(* IEC 61131-3 sources: CodesysPractice/Lessons/Lesson1/st, 7 files *)

(* ---- DUT.st ---- *)
(* =====================================================================
   对象类型 : DUT            对象名 : DUT
   项目     : Lesson1
   角色     : 全工程唯一的自定义类型表，分两个层次：
              【领域类型】Axis（一根轴）、Cmd（一条命令）—— 业务的语言；
              【报文格式】AxisInfo（PLC 发给上位机的帧）—— 线上的字节合同。
              Cmd 同时就是上行帧（命令即报文）；AxisInfo 只是输出报文，
              不是与 Axis / Cmd 并列的领域概念。

   报文布局（pack_mode=1，双端 x86/x64 小端，内存拷贝即协议）:
      Cmd    30 字节 : bType(1) bSub(1) nLen(1) aParam[3]×AxisParam(27)
      AxisParam 9 字节 : bAxis(1) rPos(4) rVel(4)
      Axis   13 字节 : rActPos(4) rTargetPos(4) rVelocity(4) xMoving(1)
      AxisInfo 45 字节 : wResult(2) nAckSeq(4) aAxis[3]×Axis(39)

   创建方法 : Application 右键 -> 添加对象 -> DUT -> 名称 DUT
              -> 类型选"结构体"（多个结构体可放在同一个 DUT 对象里）。
   粘贴方法 : 本文件整段照粘（编辑器自带的外壳整段替换）。
   ===================================================================== *)

// ==================== 领域类型 ====================

// ---- 一根轴：设定 + 实际的全部家当 ----
{attribute 'pack_mode' := '1'}
TYPE Axis :
STRUCT
    rActPos    : REAL;   // 实际位置
    rTargetPos : REAL;   // 目标位置（最近一次 MoveTo 的设定）
    rVelocity  : REAL;   // 速度（最近一次 MoveTo 的设定）
    xMoving    : BOOL;   // TRUE=运动中，FALSE=Idle
END_STRUCT
END_TYPE

// ---- 一路轴参数（CMD_CONTENT 的元素）：轴号 + 位置 + 速度 ----
{attribute 'pack_mode' := '1'}
TYPE AxisParam :
STRUCT
    bAxis : BYTE;    // 轴号：1=X 2=Y 3=Z（即 GVL.aAxis 的下标）
    rPos  : REAL;    // MOVE 目标位置（STOP 时不用）
    rVel  : REAL;    // MOVE 速度，必须 > 0（STOP 时不用）
END_STRUCT
END_TYPE

// ---- 一条命令：上位机 -> PLC，同时就是上行帧，30 字节 ----
// 分层：命令头(bType) + 子命令(bSub) + 参数数组(aParam + 有效个数 nLen)。
// 一帧可携带多路轴参数，一次命令多根轴；每路自带轴号，顺序无关。
{attribute 'pack_mode' := '1'}
TYPE Cmd :
STRUCT
    bType  : BYTE;                      // 命令头：取值见 GVL 常量 CMD_MOVE / CMD_STOP
    bSub   : BYTE;                      // 子命令：预留，现填 0（将来如 MOVE 的绝对/相对）
    nLen   : BYTE;                      // aParam 里的有效路数：1..3
    aParam : ARRAY[1..3] OF AxisParam;  // 参数数组，只有前 nLen 路有效
END_STRUCT
END_TYPE

// ==================== 报文格式 ====================

// ---- 汇报帧：PLC -> 上位机，45 字节 ----
// 只是"PLC 发出的电报"：最近一条命令的结果 + 三轴现状。
// 回执序号变化立即发一帧，否则每 200ms 发一帧 —— 两种场合发同一个结构。
{attribute 'pack_mode' := '1'}
TYPE AxisInfo :
STRUCT
    wResult : WORD;                  // 最近一条命令的结果码（0=OK，其余见 GVL 结果码）
    nAckSeq : UDINT;                 // 回执序号：上位机靠它的变化识别"新回执"
    aAxis   : ARRAY[1..3] OF Axis;   // 三轴现状
END_STRUCT
END_TYPE

(* ---- GVL.st ---- *)
(* =====================================================================
   对象类型 : GVL            对象名 : GVL
   项目     : Lesson1
   角色     : 全工程唯一的全局变量表，分两层：
              【领域数据】三根轴、当前命令 —— 业务的语言；
              【配套机制】命令的处理结果、跨任务序号握手 —— 实现细节。
              纪律：一个变量只有一个写者。
   创建方法 : Application 右键 -> 添加对象 -> 全局变量列表（GVL）-> 名称 GVL。
   粘贴方法 : 本文件整段照粘（编辑器自带的 VAR_GLOBAL...END_VAR 外壳整段替换，
              注意本文件有两个 VAR_GLOBAL 块，都要粘进去）。
   ===================================================================== *)
{attribute 'qualified_only'}
VAR_GLOBAL CONSTANT
    // ==== 命令字：Cmd.bType 的合法取值 ====
    CMD_MOVE    : BYTE := 1;
    CMD_STOP    : BYTE := 2;

    // ==== 结果码：全工程唯一出处。AxisInfo.wResult 就是这里的值，
    //      上位机按码判错 ====
    OK          : WORD := 0;      // 成功
    UNKNOWN_CMD : WORD := 1001;   // 命令字不认识（只认 CMD_MOVE / CMD_STOP）
    BAD_AXIS    : WORD := 1002;   // 轴号不是 1..3
    BAD_PARAM   : WORD := 1003;   // 参数非法（如速度 <= 0）
    SOCK_CREATE : WORD := 9001;   // 监听套接字创建失败
    SOCK_BIND   : WORD := 9002;   // 端口绑定失败（最常见：端口被占用）
    SOCK_LISTEN : WORD := 9003;   // listen 失败
END_VAR

VAR_GLOBAL
    // ==== 领域数据 ====
    aAxis   : ARRAY[1..3] OF Axis;  // 三根轴：下标即轴号 1=X / 2=Y / 3=Z
                                    // （MainTask 写，CommTask 读去组 AxisInfo）
    stCmd   : Cmd;                  // 当前命令（CommTask 收帧写入，MainTask 处理）

    // ==== stCmd 的配套机制（跨任务握手，实现细节，不是领域概念）====
    // 规则：CommTask 凑满一帧 -> stCmd 已被 FB_TcpServer 写好 -> nCmdSeq +1；
    //      MainTask 看到 nCmdSeq <> nAckSeq 就处理，处理完写 wResult、
    //      把 nAckSeq 对齐 nCmdSeq。
    // 单命令槽：上一帧没被取走时会被新帧覆盖。命令是人手速发的，骨架阶段够用；
    //          将来接自动上位机时换命令队列。
    wResult : WORD;             // stCmd 的处理结果（MainTask 写）
    nCmdSeq : UDINT := 0;       // 命令序号，CommTask 每收满一帧 +1；回绕到 0 也安全
    nAckSeq : UDINT := 0;       // 回执序号，MainTask 处理完对齐 nCmdSeq
END_VAR

(* ---- FB_CmdHandler.st ---- *)
(* =====================================================================
   对象类型 : POU（FB，语言 ST）   对象名 : FB_CmdHandler
   项目     : Lesson1
   角色     : 命令处理：解析当前命令（GVL.stCmd），分发到具体的处理者。
              它只懂协议 —— 命令字合法吗、路数合法吗、轴号合法吗；不懂业务。
              MOVE / STOP 是轴命令，业务在轴的方法（MoveTo / Stop）里；
              将来命令集合扩张（新 bType、bSub 取值、非轴命令）时，
              新增对应的处理类、加分支即可，本类结构不变。
              多路命令采用两遍法：先整体校验，再逐路执行 ——
              要么全执行，要么全不执行，不存在"动了一半"。
   协议     : bType = GVL.CMD_MOVE / GVL.CMD_STOP；bSub 预留填 0
              nLen  = 1..3（aParam 的有效路数）
              每路：bAxis = 1..3；MOVE 要求 rVel > 0（轴自己也会再判一道）
   创建方法 : Application 右键 -> 添加对象 -> POU -> 名称 FB_CmdHandler
              -> 类型选"功能块"（Function Block）-> 实现语言选 ST。
   粘贴方法 : 跳过下面第一行对象头（FUNCTION_BLOCK xxx），声明区（各 VAR 块）
              粘到编辑器上半部，"实现区"分隔线以下的内容粘到下半部。
   ===================================================================== *)
FUNCTION_BLOCK FB_CmdHandler
VAR_INPUT
    stCmd   : Cmd;                          // 待处理的当前命令
END_VAR
VAR_IN_OUT
    aAxis   : ARRAY[1..3] OF FB_SimAxis;    // 分发目标：命令最终作用在轴上
END_VAR
VAR_OUTPUT
    wResult : WORD;                         // 处理结果码：GVL.OK 或结果码
END_VAR
VAR
    i       : INT;
    nAx     : INT;
END_VAR
(* ---------------- 实现区（以下粘到 POU 编辑器下半部） ---------------- *)
// 默认成功，走到哪步出错在哪步盖结果码
wResult := GVL.OK;

// --- 命令字（协议级校验）---
IF (stCmd.bType <> GVL.CMD_MOVE) AND (stCmd.bType <> GVL.CMD_STOP) THEN
    wResult := GVL.UNKNOWN_CMD;
    RETURN;
END_IF

// --- 有效路数 ---
IF (stCmd.nLen < 1) OR (stCmd.nLen > 3) THEN
    wResult := GVL.BAD_PARAM;
    RETURN;
END_IF

// --- 第一遍：整体校验全部路数（轴号；MOVE 还要速度 > 0）---
// 任何一路非法 -> 整体拒绝，一路都不执行
FOR i := 1 TO TO_INT(stCmd.nLen) DO
    IF (stCmd.aParam[i].bAxis < 1) OR (stCmd.aParam[i].bAxis > 3) THEN
        wResult := GVL.BAD_AXIS;
        RETURN;
    END_IF
    IF (stCmd.bType = GVL.CMD_MOVE) AND (stCmd.aParam[i].rVel <= 0) THEN
        wResult := GVL.BAD_PARAM;
        RETURN;
    END_IF
END_FOR

// --- 第二遍：逐路分发执行（校验已过，此处必成功）---
FOR i := 1 TO TO_INT(stCmd.nLen) DO
    nAx := TO_INT(stCmd.aParam[i].bAxis);
    CASE stCmd.bType OF
        GVL.CMD_MOVE:
            wResult := aAxis[nAx].MoveTo(stCmd.aParam[i].rPos,
                                         stCmd.aParam[i].rVel);
        GVL.CMD_STOP:
            aAxis[nAx].Stop();
    END_CASE
END_FOR

(* ---- FB_SimAxis.st ---- *)
(* =====================================================================
   对象类型 : POU（FB，语言 ST，带 2 个方法）   对象名 : FB_SimAxis
   项目     : Lesson1
   角色     : 仿真轴：恒速点位 + 立即停止。轴是对象：
              行为是方法（MoveTo / Stop），本体每周期只做积分更新。
              参数合法性（速度 > 0）由轴自己判 —— 那是轴的业务，
              不是协议的事。换真轴时方法内部改调 MC_MoveAbsolute /
              MC_Stop，调用侧零改动。
   为什么自写而不上 SoftMotion：架子阶段要的是"一定跑得起来"。虚拟轴也要
              装 SoftMotion、配三组轴对象，把通信架子的首跑拖进运动控制
              的泥潭；接口设计好，后面换芯不动架。
   创建方法 : Application 右键 -> 添加对象 -> POU -> 名称 FB_SimAxis
              -> 类型选"功能块"（Function Block）-> 实现语言选 ST。
              然后右键 FB_SimAxis -> 添加对象 -> 方法（Method）：
              名 MoveTo、返回类型 WORD、语言 ST；名 Stop、无返回类型、语言 ST。
   粘贴方法 : FB 本体：跳过第一行对象头，VAR 块粘到上半部，"本体实现区"
              分隔线以下粘到下半部。★ 两个 METHOD 分隔线以下的内容
              **不要粘进 FB**（FB 里出现 METHOD 关键字会报"未预期的语句"）——
              方法是挂在 FB 下的独立子对象，逐节粘进对应的方法编辑器：
              跳过该节的 METHOD 对象头（IDE 按创建对话框自动生成），
              VAR 块粘上半部，实现粘下半部。
   ===================================================================== *)
FUNCTION_BLOCK FB_SimAxis
VAR_INPUT
    rCycleTime : REAL := 0.01;   // 调用任务的周期（秒），由调用方按任务配置填
END_VAR
VAR_OUTPUT
    rActPos    : REAL;           // 实际位置
    rTargetPos : REAL;           // 目标位置（最近一次 MoveTo 的设定）
    rVelocity  : REAL;           // 速度（最近一次 MoveTo 的设定）
    xMoving    : BOOL;           // TRUE=运动中
END_VAR
VAR
    rDir  : REAL := 1.0;         // 运动方向（+1/-1），MoveTo 时设定
    rStep : REAL;                // 本周期的步进量
END_VAR
(* ---------------- 本体实现区（粘到 FB 编辑器下半部） ---------------- *)
// 本体每周期只做一件事：恒速积分，到点钳位（防过冲）
IF xMoving THEN
    rStep := rVelocity * rCycleTime * rDir;
    IF ((rDir > 0) AND ((rActPos + rStep) >= rTargetPos)) OR
       ((rDir < 0) AND ((rActPos + rStep) <= rTargetPos)) THEN
        rActPos := rTargetPos;
        xMoving := FALSE;                        // 到位
    ELSE
        rActPos := rActPos + rStep;
    END_IF
END_IF

(* ============ METHOD MoveTo（独立子对象，不要粘进 FB 本体！） ============ *)
METHOD MoveTo : WORD
VAR_INPUT
    rPos : REAL;   // 目标位置
    rVel : REAL;   // 速度，必须 > 0
END_VAR
(* ---- MoveTo 实现 ---- *)
// 返回值是 GVL 结果码；运动中再来 = 改目标
MoveTo := GVL.OK;
IF rVel <= 0 THEN
    MoveTo := GVL.BAD_PARAM;
    RETURN;
END_IF
rTargetPos := rPos;
rVelocity  := rVel;
IF rTargetPos = rActPos THEN
    xMoving := FALSE;                            // 已经在点上
ELSE
    xMoving := TRUE;
    IF rTargetPos > rActPos THEN
        rDir := 1.0;
    ELSE
        rDir := -1.0;
    END_IF
END_IF

(* ============ METHOD Stop（独立子对象，不要粘进 FB 本体！） ============ *)
METHOD Stop
(* ---- Stop 实现 ---- *)
// 立即停止
xMoving := FALSE;

(* ---- FB_TcpServer.st ---- *)
(* =====================================================================
   对象类型 : POU（FB，语言 ST）   对象名 : FB_TcpServer
   项目     : Lesson1
   运行目标 : CODESYS Control Win V3 x64（64 位！）
   角色     : TCP 服务器封装（SysSocket 库）：监听 -> 接单客户端 ->
              收字节凑成定长帧 / 把一帧发出去。协议内容它一概不懂，
              只认识帧长度 —— 这就是"协议层"和"通道层"的分界。
   纪律     : 全部 socket 调用都是非阻塞的（FIONBIO），
              绝不许把 CommTask 卡死在对端的沉默上。
   注意     : 定长帧没有同步头 —— 对端发来的字节数一旦错位就会永久错位。
              骨架双方都是自己人（配套上位机），不处理；接陌生对端时
              要加帧头 + 长度 + CRC（已记入项目 README 的扩展点）。

   —— 为什么用 SysSocket 而不是 SysSockets23 ——
   旧的 SysSockets23（3.5.13.0）是 32 位专用库，在 x64 设备上编译直接报
   C0338（该库不支持 64 位应用程序）。现役的 **SysSocket**（3.5.19.0）
   是 32/64 位通用版，本文件按它的实际签名编写。

   创建方法 : Application 右键 -> 添加对象 -> POU -> 名称 FB_TcpServer
              -> 类型选"功能块"（Function Block）-> 实现语言选 ST。
   库       : Library Manager -> Add Library -> 搜 syssocket -> 选 **SysSocket**
              （3.5.19.0）。★ 不要选 SysSocket23（32 位专用），
              也不要选 SysSocket2（另一套已废弃的 2.x 接口）。
              加好后把旧的 SysSockets23 从 Library Manager 里删掉。
   粘贴方法 : 跳过下面第一行对象头（FUNCTION_BLOCK xxx），声明区（各 VAR 块）
              粘到编辑器上半部，"实现区"分隔线以下的内容粘到下半部。
   ===================================================================== *)
FUNCTION_BLOCK FB_TcpServer
VAR_INPUT
    xEnable : BOOL := TRUE;      // FALSE 时关闭连接与监听，回到空闲
    nPort   : UINT := 12000;
    pRxBuf  : POINTER TO BYTE;   // 收帧目标：凑满 nRxSize 字节 = 一帧
    nRxSize : UINT;              // 收帧长度（调用方传 SIZEOF(命令结构体)）
    pTxBuf  : POINTER TO BYTE;   // 待发的一帧
    nTxSize : UINT;              // 发帧长度
    xSend   : BOOL;              // 上升沿把 pTxBuf 指向的 nTxSize 字节发出去
END_VAR
VAR_OUTPUT
    xClientConnected : BOOL;
    xFrameReady : BOOL;          // 本周期凑满一帧（pRxBuf 内容已更新），保持一个周期
    bError      : BOOL;          // 保持型：建监听失败才置位，码见 GVL.SOCK_*
    nErrorID    : WORD;
END_VAR
VAR
    eState     : INT := 0;       // 0=空闲 / 1=监听中 / 2=已连接；不出本 FB，故不建枚举
    hListen    : RTS_IEC_HANDLE := RTS_INVALID_HANDLE;
    hClient    : RTS_IEC_HANDLE := RTS_INVALID_HANDLE;
    hNew       : RTS_IEC_HANDLE;
    sockAddr    : SOCKADDRESS;   // 本机监听地址
    sockAddrCli : SOCKADDRESS;   // accept 回写的客户端地址（内容不用，签名要指针）
    diAddrLen   : DINT;          // sockAddrCli 的长度（accept 的入/出参）
    resOp      : RTS_IEC_RESULT; // create / bind / listen / accept 的返回码
    resRecv    : RTS_IEC_RESULT; // recv 的返回码：区分"对端关闭"与"暂无数据"
    resSend    : RTS_IEC_RESULT;
    diNonBlock : DINT := 1;      // FIONBIO 参数：1 = 非阻塞
    diReuse    : DINT := 1;      // SO_REUSEADDR 参数：1 = 允许地址复用
    diRet      : __XINT;         // recv 返回值。__XINT = 平台相关整型（x64 下 64 位），
                                 // 必须用 __XINT 接，用 DINT 接在 x64 上报类型错
    diSent     : __XINT;         // send 返回值：<=0 视为发送失败（对端已死）
    diRxCnt    : INT;            // 本帧已收字节数（兼作写入偏移；指针运算用 INT 最稳）
    xBufSize   : __XINT;         // recv / send 的缓冲长度入参：类型必须和形参一致（__XINT），
                                 // 先把长度算进这个变量，实参里就不做类型转换
    xSendPrev  : BOOL;
END_VAR
VAR CONSTANT
    // SysSocket 函数的成功返回码 = 0。
    // 不直接写库常量 ERR_OK：它由库的依赖链带出，库版本一变就可能"没有定义标识符"。
    // 用本地常量最稳，语义一样。
    SOCK_OK : RTS_IEC_RESULT := 0;
    // x64 下 SysSocket 出错时返回的非法句柄是 16#FFFFFFFFFFFFFFFF
    // （Windows 的 INVALID_SOCKET），与 RTS_INVALID_HANDLE
    // （16#00000000FFFFFFFF）不相等！create / accept 拿到返回值后先归一成
    // RTS_INVALID_HANDLE，否则空 accept 会被当成接到了客户端
    // （假连接死循环：发送失败 -> 回监听 -> 又假 accept，真客户端进不来）。
    HANDLE_INVALID : RTS_IEC_HANDLE := 16#FFFFFFFFFFFFFFFF;
END_VAR
(* ---------------- 实现区（以下粘到 POU 编辑器下半部） ---------------- *)
xFrameReady := FALSE;

// --- 使能撤掉：关干净回空闲 ---
IF NOT xEnable THEN
    IF (hClient <> RTS_INVALID_HANDLE) AND (hClient <> 0) THEN
        SysSockClose(hClient);
        hClient := RTS_INVALID_HANDLE;
    END_IF
    IF (hListen <> RTS_INVALID_HANDLE) AND (hListen <> 0) THEN
        SysSockClose(hListen);
        hListen := RTS_INVALID_HANDLE;
    END_IF
    eState := 0;
    xClientConnected := FALSE;
    diRxCnt := 0;
END_IF

CASE eState OF

    // ---------------------------------------------------------------
    0:  // 空闲：建立监听
        bError := FALSE;
        nErrorID := GVL.OK;
        IF xEnable THEN
            // SysSockCreate(iAddressFamily : INT, diType : DINT, diProtocol : DINT,
            //               pResult : POINTER TO RTS_IEC_RESULT) : RTS_IEC_HANDLE
            hListen := SysSockCreate(SOCKET_AF_INET, SOCKET_STREAM, SOCKET_IPPROTO_TCP,
                                     ADR(resOp));
            IF hListen = HANDLE_INVALID THEN
                hListen := RTS_INVALID_HANDLE;   // 归一非法句柄，见 HANDLE_INVALID 注释
            END_IF
            IF (hListen = RTS_INVALID_HANDLE) OR (hListen = 0) THEN
                bError := TRUE;
                nErrorID := GVL.SOCK_CREATE;
                hListen := RTS_INVALID_HANDLE;
            ELSE
                // 非阻塞：accept / recv 没有事件时立即返回，不卡任务
                // SysSockIoctl(hSocket, diCommand : DINT, pdiParameter : POINTER TO DINT)
                SysSockIoctl(hListen, SOCKET_FIONBIO, ADR(diNonBlock));
                // 允许地址复用：调试时反复"下载/运行"不会报端口被占用（9002）
                // SysSockSetOption(hSocket, diLevel : DINT, diOption : DINT,
                //                  pdiOptionValue : POINTER TO DINT, diOptionLen : DINT)
                SysSockSetOption(hListen, SOCKET_SOL, SOCKET_SO_REUSEADDR,
                                 ADR(diReuse), SIZEOF(diReuse));

                sockAddr.sin_family      := SOCKET_AF_INET;      // INT，直接赋值，不要 TO_INT
                // 端口必须转成网络字节序；显式 WORD 转型避免 UINT->WORD 的隐式转换告警
                sockAddr.sin_port        := SysSockHtons(TO_WORD(nPort));
                sockAddr.sin_addr.ulAddr := SOCKET_INADDR_ANY;   // 0.0.0.0，本机所有网卡都接

                // SysSockBind(hSocket, pSockAddr : POINTER TO SOCKADDRESS,
                //             diSockAddrSize : DINT) : RTS_IEC_RESULT
                IF SysSockBind(hListen, ADR(sockAddr), SIZEOF(sockAddr)) <> SOCK_OK THEN
                    bError := TRUE;
                    nErrorID := GVL.SOCK_BIND;
                // SysSockListen(hSocket, diMaxConnections : DINT) : RTS_IEC_RESULT
                ELSIF SysSockListen(hListen, 1) <> SOCK_OK THEN
                    bError := TRUE;
                    nErrorID := GVL.SOCK_LISTEN;
                ELSE
                    eState := 1;
                END_IF
                IF bError THEN
                    SysSockClose(hListen);
                    hListen := RTS_INVALID_HANDLE;
                END_IF
            END_IF
        END_IF

    // ---------------------------------------------------------------
    1:  // 监听中：非阻塞 accept，接到就进已连接
        // SysSockAccept(hSocket, pSockAddr : POINTER TO SOCKADDRESS,
        //               pdiSockAddrSize : POINTER TO DINT,
        //               pResult) : RTS_IEC_HANDLE
        // 注意：x64 版不接受空指针（0），必须传真实的地址变量和长度变量
        diAddrLen := SIZEOF(sockAddrCli);
        hNew := SysSockAccept(hListen, ADR(sockAddrCli), ADR(diAddrLen), ADR(resOp));
        IF hNew = HANDLE_INVALID THEN
            hNew := RTS_INVALID_HANDLE;          // 归一非法句柄，见 HANDLE_INVALID 注释
        END_IF
        IF (hNew <> RTS_INVALID_HANDLE) AND (hNew <> 0) THEN
            hClient := hNew;
            SysSockIoctl(hClient, SOCKET_FIONBIO, ADR(diNonBlock));
            diRxCnt := 0;
            xClientConnected := TRUE;
            eState := 2;
        END_IF

    // ---------------------------------------------------------------
    2:  // 已连接：收字节凑帧 / 发一帧
        // -- 收：往调用方的帧缓冲里续字节，凑满 nRxSize 即一帧 --
        IF (pRxBuf <> 0) AND (nRxSize > 0) THEN
            // SysSockRecv(hSocket, pbyBuffer : POINTER TO BYTE, diBufferSize : __XINT,
            //             diFlags : DINT, pResult) : __XINT
            // flags 传 NONE：非阻塞由 socket 级的 FIONBIO 保证。
            // 不要传 MSG_DONTWAIT（16#8）——那是 Linux 语义，Windows 运行时下
            // 16#8 是 MSG_WAITALL，会让 recv 行为异常、读不到数据
            xBufSize := TO_INT(nRxSize) - diRxCnt;       // 本帧还缺的字节数
            diRet := SysSockRecv(hClient, pRxBuf + diRxCnt,
                                 xBufSize, SOCKET_MSG_NONE, ADR(resRecv));
            IF diRet > 0 THEN
                diRxCnt := diRxCnt + TO_INT(diRet);
                IF diRxCnt >= TO_INT(nRxSize) THEN
                    diRxCnt := 0;                        // 下一帧从头开始凑
                    xFrameReady := TRUE;
                END_IF
            ELSIF (diRet = 0) AND (resRecv = SOCK_OK) THEN
                // 收到 0 字节且无错误 = 对端正常关闭 -> 回监听态等下一个客户端；
                // 没收完的半帧随 diRxCnt 清零一起丢弃
                SysSockClose(hClient);
                hClient := RTS_INVALID_HANDLE;
                xClientConnected := FALSE;
                diRxCnt := 0;
                eState := 1;
            END_IF
            // diRet = 0 且 resRecv <> SOCK_OK：非阻塞下"暂无数据"，不是错误
        END_IF

        // -- 发：xSend 上升沿 --
        // 骨架不做短写重发：本机回环 + 一帧 21 字节，一次写不完的概率为零；
        // 将来走真实网络时必须处理短写（已记入项目 README 的扩展点）
        IF xSend AND NOT xSendPrev AND (pTxBuf <> 0) THEN
            // SysSockSend(hSocket, pbyBuffer, diBufferSize : __XINT,
            //             diFlags : DINT, pResult) : __XINT
            xBufSize := nTxSize;
            diSent := SysSockSend(hClient, pTxBuf, xBufSize, SOCKET_MSG_NONE, ADR(resSend));
            // 死连接检测（不依赖 recv 的返回码语义）：对端关闭后，
            // 头一两次 send 可能还"成功"，对端 OS 回 RST 之后 send 必失败。
            // 状态帧每 200ms 一发，所以断开最多 ~400ms 内被发现并自愈：
            // 关掉死句柄回监听态，backlog 里排队的新连接下一周期被 accept。
            // 注意：本机回环下发送缓冲永远不会满，"0=失败"不会误伤活连接。
            IF diSent <= 0 THEN
                SysSockClose(hClient);
                hClient := RTS_INVALID_HANDLE;
                xClientConnected := FALSE;
                diRxCnt := 0;
                eState := 1;
            END_IF
        END_IF

END_CASE

xSendPrev := xSend;

(* ---- PRG_Comm.st ---- *)
(* =====================================================================
   对象类型 : POU（PRG，语言 ST）  对象名 : PRG_Comm
   项目     : Lesson1
   任务     : CommTask（20 ms，优先级低于 MainTask）
   纪律     : 只收发原始帧，不认识协议内容：收帧写进 GVL.stCmd、
              回执序号变化就立即发一帧 AxisInfo、否则周期发。
              解析和执行永远是 MainTask 的事。
   创建方法 : Application 右键 -> 添加对象 -> POU -> 名称 PRG_Comm
              -> 类型选"程序"（Program）-> 实现语言选 ST。
   粘贴方法 : 跳过下面第一行对象头（PROGRAM xxx），声明区（VAR 块）粘到
              编辑器上半部，"实现区"分隔线以下的内容粘到下半部。
   ===================================================================== *)
PROGRAM PRG_Comm
VAR
    fbTcp      : FB_TcpServer;
    stAxisInfo   : AxisInfo;      // 待发的一帧（回执与周期状态共用同一个结构）
    nLastAck   : UDINT := 0;      // 上次发出帧里带的回执序号
    nStatusDiv : UINT := 0;       // 状态帧分频：20ms x 10 = 200ms 一帧
    xSend      : BOOL;
END_VAR
(* ---------------- 实现区（以下粘到 POU 编辑器下半部） ---------------- *)

// --- 1) 发送仲裁：回执优先于周期状态。一周期最多发一帧，
//        TCP 会排队不丢，状态帧晚 20ms 无碍 ---
xSend := FALSE;
IF GVL.nAckSeq <> nLastAck THEN
    nLastAck := GVL.nAckSeq;
    xSend := TRUE;
ELSE
    nStatusDiv := nStatusDiv + 1;
    IF nStatusDiv >= 10 THEN
        nStatusDiv := 0;
        xSend := TRUE;           // 无客户端时 FB_TcpServer 内部会丢弃
    END_IF
END_IF

IF xSend THEN
    stAxisInfo.wResult := GVL.wResult;   // 结果码随每一帧带出去
    stAxisInfo.nAckSeq := GVL.nAckSeq;   // 上位机靠它的变化识别新回执
    stAxisInfo.aAxis   := GVL.aAxis;
END_IF

// --- 2) 跑服务器：收到的字节直接凑进 GVL.stCmd ---
fbTcp(
    xEnable := TRUE,
    nPort   := 12000,
    pRxBuf  := ADR(GVL.stCmd),
    nRxSize := SIZEOF(Cmd),
    pTxBuf  := ADR(stAxisInfo),
    nTxSize := SIZEOF(AxisInfo),
    xSend   := xSend);

// --- 3) 凑满一帧 -> 命令序号 +1（GVL.stCmd 只允许本任务写）---
IF fbTcp.xFrameReady THEN
    GVL.nCmdSeq := GVL.nCmdSeq + 1;
END_IF

(* ---- PRG_Main.st ---- *)
(* =====================================================================
   对象类型 : POU（PRG，语言 ST）  对象名 : PRG_Main
   项目     : Lesson1
   任务     : MainTask（10 ms，优先级最高）
   纪律     : PRG 只做调度 —— 新命令交给 FB_CmdHandler 解析分发、
              周期驱动三轴、把状态发布到 GVL。
   创建方法 : Application 右键 -> 添加对象 -> POU -> 名称 PRG_Main
              -> 类型选"程序"（Program）-> 实现语言选 ST。
   粘贴方法 : 跳过下面第一行对象头（PROGRAM xxx），声明区（VAR 块）粘到
              编辑器上半部，"实现区"分隔线以下的内容粘到下半部。
   ===================================================================== *)
PROGRAM PRG_Main
VAR
    fbCmdHandler : FB_CmdHandler;
    fbAxis       : ARRAY[1..3] OF FB_SimAxis;   // 下标 = 轴号（1=X / 2=Y / 3=Z）
    i            : INT;
END_VAR
(* ---------------- 实现区（以下粘到 POU 编辑器下半部） ---------------- *)

// --- 1) 来了新命令：解析 + 分发 + 回执（接受与拒绝都回执、都回显序号）---
IF GVL.nCmdSeq <> GVL.nAckSeq THEN
    fbCmdHandler(stCmd := GVL.stCmd, aAxis := fbAxis);
    GVL.wResult := fbCmdHandler.wResult;
    GVL.nAckSeq := GVL.nCmdSeq;
END_IF

// --- 2) 周期驱动三轴，并把状态发布到 GVL（本任务唯一写者）---
FOR i := 1 TO 3 DO
    fbAxis[i](rCycleTime := 0.01);              // 与 MainTask 周期一致
    GVL.aAxis[i].rActPos    := fbAxis[i].rActPos;
    GVL.aAxis[i].rTargetPos := fbAxis[i].rTargetPos;
    GVL.aAxis[i].rVelocity  := fbAxis[i].rVelocity;
    GVL.aAxis[i].xMoving    := fbAxis[i].xMoving;
END_FOR
